{attribute 'qualified_only'}
TYPE E_Foo01 :
(
	eNoError := 0,
	eErrorA := 1,
	eErrorB := 2
);
END_TYPE

(* stored: Version 1.1.0.1, ProductVersion 3.1.4020.6
   DUT E_Foo01: Id {a4e3f45c-f592-40eb-8512-00324c08bef3} *)
